SYSTEM FLASHER_TESTR (* Remote Flasher Test System Configuration *)
  (* Standard: 61499-1 *)
  (* Version 0.2, 2007-11-07, JHC, Holobloc Inc, Re-implemented as per FLASHER_TESTD. *)
  (* Version 0.1, 2006-10-27, JHC, Holobloc Inc, Added multiple CLIENT/SERVERs. *)
  (* Version 0.0, 2006-10-25, JHC, Holobloc Inc, Copied from FLASHERT_TESTR to fb.rt.doc. *)
  DEVICE CTL_PANEL : FRAME_DEVICE(BOUNDS := [50,100,350,100], GRID := [1,1])
    RESOURCE RES1 : PANEL_RESOURCE
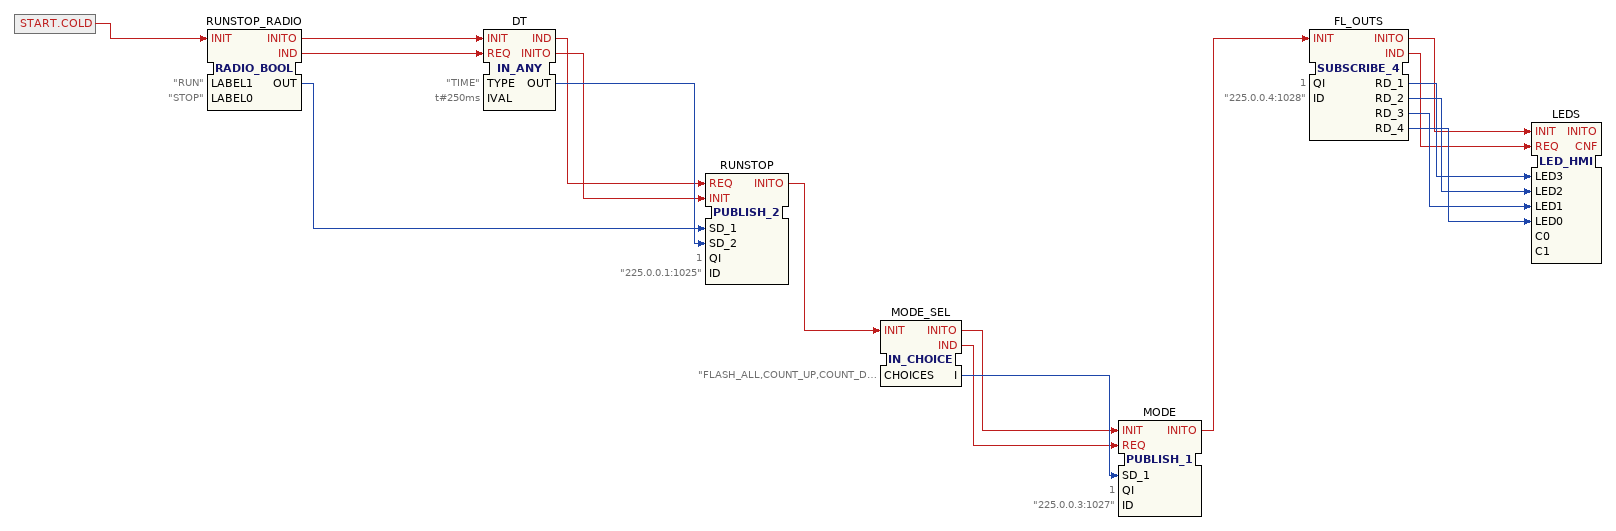
      FBS
        RUNSTOP_RADIO : RADIO_BOOL(LABEL1 := "RUN", LABEL0 := "STOP");
        MODE_SEL : IN_CHOICE(CHOICES := "FLASH_ALL,COUNT_UP,COUNT_DOWN,CHASE_UP,CHASE_DOWN");
        DT : IN_ANY(TYPE := "TIME", IVAL := t#250ms);
        RUNSTOP : PUBLISH_2(QI := 1, ID := "225.0.0.1:1025");
        MODE : PUBLISH_1(QI := 1, ID := "225.0.0.3:1027");
        LEDS : LED_HMI;
        FL_OUTS : SUBSCRIBE_4(QI := 1, ID := "225.0.0.4:1028");
      END_FBS
      EVENT_CONNECTIONS
        START.COLD TO RUNSTOP_RADIO.INIT;
        RUNSTOP_RADIO.INITO TO DT.INIT;
        RUNSTOP_RADIO.IND TO DT.REQ;
        DT.IND TO RUNSTOP.REQ;
        DT.INITO TO RUNSTOP.INIT;
        RUNSTOP.INITO TO MODE_SEL.INIT;
        MODE_SEL.INITO TO MODE.INIT;
        MODE_SEL.IND TO MODE.REQ;
        MODE.INITO TO FL_OUTS.INIT;
        FL_OUTS.INITO TO LEDS.INIT;
        FL_OUTS.IND TO LEDS.REQ;
      END_CONNECTIONS
      DATA_CONNECTIONS
        RUNSTOP_RADIO.OUT TO RUNSTOP.SD_1;
        DT.OUT TO RUNSTOP.SD_2;
        MODE_SEL.I TO MODE.SD_1;
        FL_OUTS.RD_1 TO LEDS.LED3;
        FL_OUTS.RD_2 TO LEDS.LED2;
        FL_OUTS.RD_3 TO LEDS.LED1;
        FL_OUTS.RD_4 TO LEDS.LED0;
      END_CONNECTIONS
    END_RESOURCE
  END_DEVICE
  DEVICE FLASHER : RMT_DEV
    RESOURCE MGR : RMT_RES
    END_RESOURCE
    RESOURCE RES1 : EMB_RES
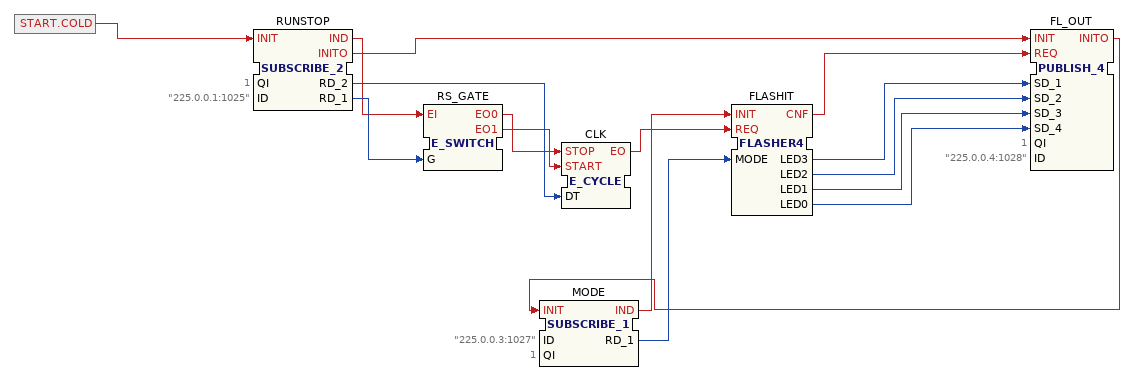
      FBS
        CLK : E_CYCLE;
        FLASHIT : FLASHER4;
        RUNSTOP : SUBSCRIBE_2(QI := 1, ID := "225.0.0.1:1025");
        RS_GATE : E_SWITCH;
        MODE : SUBSCRIBE_1(ID := "225.0.0.3:1027", QI := 1);
        FL_OUT : PUBLISH_4(QI := 1, ID := "225.0.0.4:1028");
      END_FBS
      EVENT_CONNECTIONS
        CLK.EO TO FLASHIT.REQ;
        START.COLD TO RUNSTOP.INIT;
        RUNSTOP.IND TO RS_GATE.EI;
        MODE.IND TO FLASHIT.INIT;
        RS_GATE.EO0 TO CLK.STOP;
        RS_GATE.EO1 TO CLK.START;
        RUNSTOP.INITO TO FL_OUT.INIT;
        FLASHIT.CNF TO FL_OUT.REQ;
        FL_OUT.INITO TO MODE.INIT;
      END_CONNECTIONS
      DATA_CONNECTIONS
        RUNSTOP.RD_2 TO CLK.DT;
        RUNSTOP.RD_1 TO RS_GATE.G;
        MODE.RD_1 TO FLASHIT.MODE;
        FLASHIT.LED3 TO FL_OUT.SD_1;
        FLASHIT.LED2 TO FL_OUT.SD_2;
        FLASHIT.LED1 TO FL_OUT.SD_3;
        FLASHIT.LED0 TO FL_OUT.SD_4;
      END_CONNECTIONS
    END_RESOURCE
  END_DEVICE
END_SYSTEM
